ABB RobotStudio station: Abb_Robo_Challenge.rspag

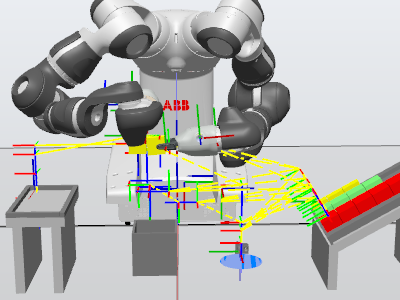
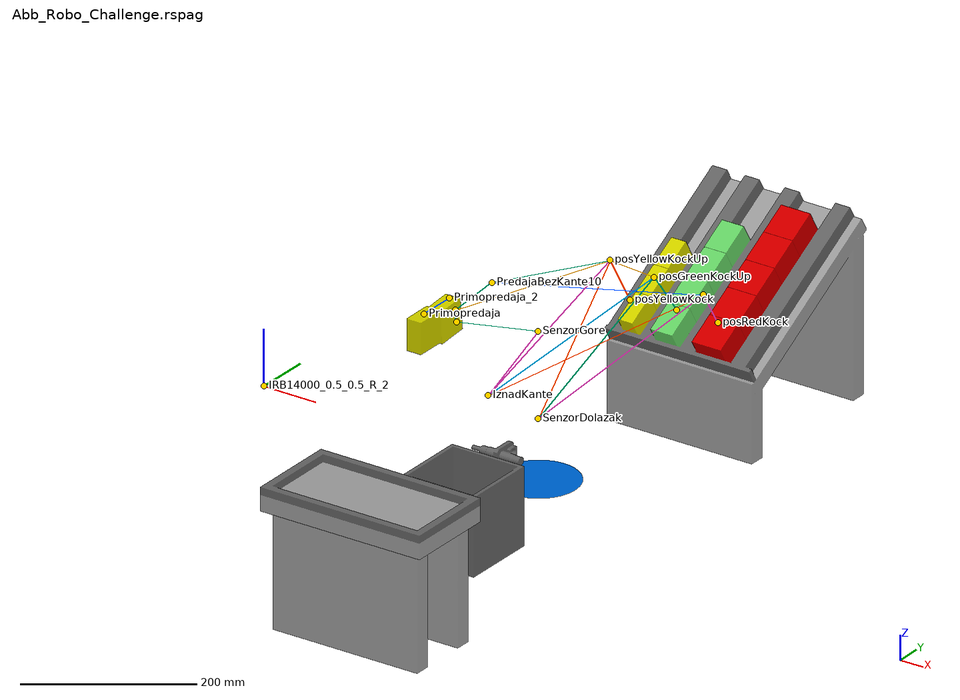
[picture v1: parts stored in the station drawn from their meshes, with robot base, taught points and paths (robot models come from the ABB library and are not in the file)]
--- station ---
Station Solution3 (saved by RobotStudio 22.3.10190.2)
Controller IRB14000, task T_ROB_L: task frame (RAPID world) sits at (0, 0, 100) mm in the station
Controller IRB14000, task T_ROB_R: task frame (RAPID world) sits at (0, 0, 100) mm in the station
Controller IRB14000
  mechanical unit ROB_R: IRB14000_0.5_0.5_R_2, 6 joints, base frame (0, 0, 0) mm
  mechanical unit ROB_R_7: IRB14000_0.5_0.5_R_2, 1 joints, base frame (0, 0, 0) mm
  mechanical unit ROB_L: IRB14000_0.5_0.5_L_2, 6 joints, base frame (0, 0, 0) mm
  mechanical unit ROB_L_7: IRB14000_0.5_0.5_L_2, 1 joints, base frame (0, 0, 0) mm
Layout (positions relative to the parent item):
  - Smart_Gripper_Servo_One_Vacuum_Fingers [mechanism, from Tools\ABB_Smart_Gripper_Servo_One_Vacuum_Fingers.rslib] at (280.99, 90.09, 293.14) mm, rotated rx 94.8 ry -1.33 rz -0.03 deg; joint values [0.0203] (rad or m)
  - Smart_Gripper_Servo_One_Vacuum_Camera_Fingers [mechanism, from Tools\ABB_Smart_Gripper_Servo_One_Vacuum_Camera_Fingers.rslib] at (319.77, -68.88, 368.32) mm, rotated rx 40.81 ry 90 rz -139.19 deg; joint values [0] (rad or m)
  - Senzor_Metala [part] at (250, 150, 15) mm, rotated rx 0 ry 0 rz 180 deg, size 65 x 32 x 27 mm
  - Mesto za testiranje [part] at (275, 150, 0) mm, size 100 x 99.5 x 0 mm
  - Rampa sa kutijama [graphiccomponentgroup]
    - Part_20 [part] at (374.5, 471.2, 184.6) mm, rotated rx 30 ry 0 rz 0 deg, size 40 x 40 x 40 mm
    - Part_1 [part] at (250, 320, 0) mm, size 200 x 20 x 100 mm
    - Part_2 [part] at (250, 520, 0) mm, size 200 x 20 x 200 mm
    - Part_3 [part], size 200 x 226.5 x 142.3 mm
    - Part_4 [part], size 200 x 14.3 x 19.8 mm
    - Part_5 [part], size 20 x 217.8 x 137.3 mm
    - Part_6 [part] at (45, 0, 0) mm, size 20 x 217.8 x 137.3 mm
    - Part_7 [part] at (100, 0, 0) mm, size 20 x 217.8 x 137.3 mm
    - Part_8 [part] at (170, 0, 0) mm, size 20 x 217.8 x 137.3 mm
    - Part_10 [part] at (292.5, 364.68, 123.1) mm, rotated rx 30 ry 0 rz 0 deg, size 20 x 40 x 40 mm
    - Part_11 [part] at (292.5, 400.18, 143.6) mm, rotated rx 30 ry 0 rz 0 deg, size 20 x 40 x 40 mm
    - Part_12 [part] at (317.5, 329.17, 102.6) mm, rotated rx 30 ry 0 rz 0 deg, size 30 x 40 x 40 mm
    - Part_13 [part] at (317.5, 364.68, 123.1) mm, rotated rx 30 ry 0 rz 0 deg, size 30 x 40 x 40 mm
    - Part_14 [part] at (317.5, 400.18, 143.6) mm, rotated rx 30 ry 0 rz 0 deg, size 30 x 40 x 40 mm
    - Part_15 [part] at (374.5, 329.17, 102.6) mm, rotated rx 30 ry 0 rz 0 deg, size 40 x 40 x 40 mm
    - Part_16 [part] at (374.5, 364.68, 123.1) mm, rotated rx 30 ry 0 rz 0 deg, size 40 x 40 x 40 mm
    - Part_17 [part] at (374.5, 400.18, 143.6) mm, rotated rx 30 ry 0 rz 0 deg, size 40 x 40 x 40 mm
    - Part_18 [part] at (317.5, 435.69, 164.1) mm, rotated rx 30 ry 0 rz 0 deg, size 30 x 40 x 40 mm
    - Part_19 [part] at (374.5, 435.69, 164.1) mm, rotated rx 30 ry 0 rz 0 deg, size 40 x 40 x 40 mm
    - Part_9 [part] at (290.75, -67.71, 300.19) mm, rotated rx -85.2 ry -1.33 rz -0.03 deg, size 20 x 40 x 40 mm
  - Paleta [graphiccomponentgroup]
    - Part_31 [part] at (450, -340, 170) mm, size 10 x 100 x 10 mm
    - Part_21 [part] at (250, -340, 0) mm, size 200 x 20 x 150 mm
    - Part_22 [part] at (250, -260, 0) mm, size 200 x 20 x 150 mm
    - Part_25 [part] at (240, -350, 170) mm, size 220 x 10 x 10 mm
    - Part_26 [part] at (240, -240, 170) mm, size 220 x 10 x 10 mm
    - Part_27 [part] at (240, -350, 150) mm, size 220 x 120 x 20 mm
    - Part_28 [part] at (240, -340, 170) mm, size 10 x 100 x 10 mm
  - Mesto za odlaganje [part], size 100 x 100 x 100 mm
  - Part_23 [part] at (292.5, 329.17, 102.6) mm, rotated rx 30 ry 0 rz 0 deg, size 20 x 40 x 40 mm
  - Pomocni_Desni [part] at (292.31, -67.5, 304.23) mm, rotated rx 180 ry 0 rz 0 deg, size 20 x 40 x 40 mm
  - IRB14000_0.5_0.5_2 [mechanism, from Robots\IRB14000_0.5_0.5__01.rslib] at (0, 0, 100) mm
  - IRB14000_0.5_0.5_R_2 [mechanism, from Robots\IRB14000_0.5_0.5__01.rslib] at (0, 0, 100) mm; joint values [1.4853, -1.6274, -1.2622, 0.7026, -0.8535, 2.2173, -1.4411] (rad or m)
  - IRB14000_0.5_0.5_L_2 [mechanism, from Robots\IRB14000_0.5_0.5__01.rslib] at (0, 0, 100) mm; joint values [-1.2905, -2.4868, 1.2641, 0.7988, -4.7194, 1.3107, 3.1478] (rad or m)
Attachment: Part_8 is attached to Part_7
Attachment: Part_7 is attached to Part_6
Attachment: Part_6 is attached to Part_5
Attachment: Part_5 is attached to Part_4
Attachment: Part_4 is attached to Part_3
Attachment: Part_3 is attached to Part_2
Attachment: Part_2 is attached to Part_1
Attachment: Part_10 is attached to Part_4
Attachment: Part_11 is attached to Part_4
Attachment: Part_12 is attached to Part_4
Attachment: Part_13 is attached to Part_4
Attachment: Part_14 is attached to Part_4
Attachment: Part_15 is attached to Part_4
Attachment: Part_16 is attached to Part_4
Attachment: Part_17 is attached to Part_4
Attachment: Part_18 is attached to Part_4
Attachment: Part_19 is attached to Part_4
Attachment: Part_20 is attached to Part_4
Attachment: Part_31 is attached to Part_28
Attachment: Part_28 is attached to Part_26
Attachment: Part_26 is attached to Part_25
Attachment: Part_25 is attached to Part_27
Attachment: Part_27 is attached to Part_22
Attachment: Part_22 is attached to Part_21
Attachment: Part_9 is attached to Smart_Gripper_Servo_One_Vacuum_Fingers / DownFinger
Attachment: Pomocni_Desni is attached to Pneumatic
Attachment: Smart_Gripper_Servo_One_Vacuum_Camera_Fingers is attached to IRB14000_0.5_0.5_R_2 / Link7
Attachment: Smart_Gripper_Servo_One_Vacuum_Fingers is attached to IRB14000_0.5_0.5_L_2 / Link7
Targets, tools, work objects and paths stored in the station and not in the controller backup, written as RAPID:
! task T_ROB_R
MODULE PROGRAM_R
  VAR syncident sync1;
  VAR syncident sync2;
  VAR syncident sync3;
ENDMODULE

! task T_ROB_L
MODULE PROGRAM_L
  VAR syncident sync1;
  VAR syncident sync2;
  VAR syncident sync3;
ENDMODULE

! task T_ROB_R
MODULE PROGRAM_R
  VAR syncident sync1;
  VAR syncident sync2;
ENDMODULE

! task T_ROB_L
MODULE PROGRAM_L
  VAR syncident sync1;
  VAR syncident sync2;
ENDMODULE


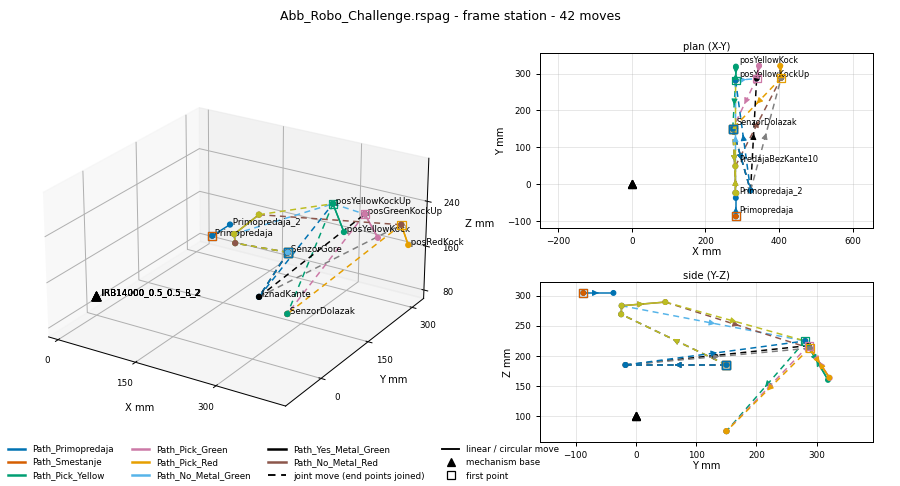
[picture p0: tool path of Abb_Robo_Challenge.rspag in frame station, 42 of 45 moves have a stored position in this frame; points joined in program order, loops and branches not executed]
--- Backups/IRB14000/RAPID/TASK1/PROGMOD/CalibData.mod ---
MODULE CalibData
    PERS tooldata Servo:=[TRUE,[[0,0,114.2],[1,0,0,0]],[0.24,[8.2,12.5,48.1],[1,0,0,0],0.00022,0.00024,0.00009]];
    PERS tooldata VaccumOne:=[TRUE,[[63.5,18.5,37.5],[0.707106781,0,0.707106781,0]],[0.24,[8.2,12.5,48.1],[1,0,0,0],0.00022,0.00024,0.00009]];
    PERS tooldata Camera:=[TRUE,[[-7.3,28.3,35.1],[0.5,-0.5,0.5,0.5]],[0.24,[8.2,12.5,48.1],[1,0,0,0],0.00022,0.00024,0.00009]];
    PERS wobjdata woKantaR:=[FALSE,TRUE,"",[[282.386,-62.26,79.768],[0.707106781,-0.707106781,0,0]],[[0,0,0],[1,0,0,0]]];
    PERS wobjdata woPreuzmi:=[FALSE,TRUE,"",[[282.386,102.74,79.768],[0.707106781,-0.707106781,0,0]],[[0,0,0],[1,0,0,0]]];
    PERS wobjdata woPaleta:=[FALSE,TRUE,"",[[250,-330.604465451,70],[1,0,0,0]],[[0,0,0],[1,0,0,0]]];
ENDMODULE

--- Backups/IRB14000/RAPID/TASK1/PROGMOD/Module1.mod ---
MODULE Module1
    PERS num br_duzina;
    PERS num br_visina;
    PERS num pomeraj;



       !  !!!!!!!!!!!!!!!!!!!!!!!!!!!!!!!!

    CONST robtarget posHome:=[[54.845252741,-184.443859011,238.96369283],[0.12531745,-0.225816146,-0.031964186,-0.965546941],[0,0,0,4],[-101.964427132,9E+09,9E+09,9E+09,9E+09,9E+09]];
    CONST robtarget posKodKante:=[[0,-100,-20],[1,0,0,0],[0,0,0,0],[-101.964427132,9E+09,9E+09,9E+09,9E+09,9E+09]];
    CONST robtarget posKodKante_3:=[[0,0,-20],[1,0,0,0],[0,0,0,0],[-101.964427132,9E+09,9E+09,9E+09,9E+09,9E+09]];
    CONST robtarget posKodKante_2:=[[0,0,0],[1,0,0,0],[0,0,0,0],[-101.964427132,9E+09,9E+09,9E+09,9E+09,9E+09]];
    CONST robtarget posTranzicija:=[[-0.118930441,-20.052950344,-210.115205223],[1,-0.000000095,-0.000000108,0.000000158],[1,-1,2,4],[-147.412404821,9E+09,9E+09,9E+09,9E+09,9E+09]];
    CONST robtarget posIznadSenzora:=[[-8.495,34.489,-98.444458216],[1,0,0,0],[1,-1,2,4],[-147.412404821,9E+09,9E+09,9E+09,9E+09,9E+09]];
    CONST robtarget posTranzicija_2:=[[-0.118939501,-5.052946544,-190.115208073],[1,-0.000000095,-0.000000108,0.000000158],[1,-1,2,4],[-147.412404821,9E+09,9E+09,9E+09,9E+09,9E+09]];

    VAR robtarget posTranzicija_3:=[[-0.118914221,-85.052946544,-170.115192873],[0.500000023,-0.500000086,0.49999982,0.500000072],[1,-1,-1,4],[-147.412404821,9E+09,9E+09,9E+09,9E+09,9E+09]];
    VAR robtarget poz_iznad_palete_2:=[[20,9.582041834,90],[0,-0.707106781,0.707106781,0],[0,0,-2,4],[-170.196454308,9E+09,9E+09,9E+09,9E+09,9E+09]];
    VAR robtarget poz_iznad_palete:=[[20.00,9.99,-12.75],[2.11141E-05,0.707095,-0.707119,-9.2686E-07],[1,0,-2,4],[-170.196,9E+09,9E+09,9E+09,9E+09,9E+09]];
    CONST robtarget Primopredaja:=[[-0.118901581,-125.052946544,-190.115185273],[0.707106714,-0.707106848,-0.000000188,0.000000035],[1,-1,-1,4],[-147.412404821,9E+09,9E+09,9E+09,9E+09,9E+09]];
    CONST robtarget Primopredaja_2:=[[-0.118912401,-125.052956019,-140.115185273],[0.707106714,-0.707106848,-0.000000188,0.000000035],[1,-1,-1,4],[-147.412404821,9E+09,9E+09,9E+09,9E+09,9E+09]];


    PROC Path_Primopredaja()

        MoveJ Primopredaja,v500,z50,VaccumOne\WObj:=woPreuzmi;
        MoveL Primopredaja_2,v50,fine,VaccumOne\WObj:=woPreuzmi;
        g_VacuumOn1;
        WaitSyncTask \InPos, sync1,task_list;


        WaitSyncTask sync2,task_list;
        WaitTime\InPos,0.1;
        WaitSyncTask sync3,task_list;

    ENDPROC
    PROC Path_Smestanje()
        poz_iznad_palete_2:=[[20+br_duzina*43,9.99+pomeraj,90+br_visina*42],[0,-0.707106781,0.707106781,0],[0,0,-2,4],[-170.196454308,9E+09,9E+09,9E+09,9E+09,9E+09]];
        !poz_iznad_palete:=[[20+br_duzina*40,10+pomeraj,45+br_visina*40],[0,-0.707106781,0.707106781,0],[1,0,-2,4],[-170.196454308,9E+09,9E+09,9E+09,9E+09,9E+09]];
        poz_iznad_palete:=[[20.00+br_duzina*43,9.99+pomeraj,-12.75+br_visina*42],[2.11141E-05,0.707095,-0.707119,-9.2686E-07],[1,0,-2,4],[-170.196,9E+09,9E+09,9E+09,9E+09,9E+09]];
        posTranzicija_3:=[[-0.118914221,-85.052946544,-170.115192873+br_visina*40],[0.500000023,-0.500000086,0.49999982,0.500000072],[1,-1,-1,4],[-147.412404821,9E+09,9E+09,9E+09,9E+09,9E+09]];


        MoveL poz_iznad_palete_2,v500,fine,VaccumOne\WObj:=woPaleta;
        MoveL poz_iznad_palete,v50,fine,VaccumOne\WObj:=woPaleta;
        WaitTime \InPos, 0.1;
        g_VacuumOff1;
        MoveL poz_iznad_palete_2,v100,fine,VaccumOne\WObj:=woPaleta;
        MoveL Primopredaja,v500,z100,VaccumOne\WObj:=woPreuzmi;
    ENDPROC
ENDMODULE

--- Backups/IRB14000/RAPID/TASK1/PROGMOD/PROGRAM_R.mod ---
MODULE PROGRAM_R

    PERS num IsMetal;
    VAR syncident sync1;
    PERS tasks task_list{2}:=[["T_ROB_L"], ["T_ROB_R"]];
    VAR syncident sync2;
    VAR syncident sync3;
    PERS bool radi;

    PROC main()
        g_Init;
        WHILE radi  DO
            Path_Primopredaja;
            IF IsMetal = 1 THEN
                g_VacuumOff1;
            ELSE
                Path_Smestanje;
            ENDIF

        ENDWHILE
    ENDPROC
ENDMODULE

--- Backups/IRB14000/RAPID/TASK2/PROGMOD/CalibData.mod ---
MODULE CalibData
    PERS tooldata Servo:=[TRUE,[[0,0,114.2],[1,0,0,0]],[0.226,[8.9,12.3,48.7],[1,0,0,0],0.00021,0.00024,0.00009]];
    PERS tooldata VaccumOne:=[TRUE,[[63.5,18.5,37.5],[0.707106781,0,0.707106781,0]],[0.226,[8.9,12.3,48.7],[1,0,0,0],0.00021,0.00024,0.00009]];
    PERS wobjdata woYellow:=[FALSE,TRUE,"",[[282.5,326.49,47.239],[0,1,0,0]],[[0,0,0],[1,0,0,0]]];
    PERS wobjdata woSenzor:=[FALSE,TRUE,"",[[250,150,-85],[0,1,0,0]],[[0,0,0],[1,0,0,0]]];
ENDMODULE

--- Backups/IRB14000/RAPID/TASK2/PROGMOD/Module1.mod ---
MODULE Module1

    PERS num IsMetal;

    CONST robtarget posHome:=[[89.387946423,156.622117957,147.913470217],[0.066010726,0.842420918,-0.111214912,0.523068661],[0,0,0,4],[101.964427132,9E+09,9E+09,9E+09,9E+09,9E+09]];
    CONST robtarget posYellowKockRanije:=[[0,18.749999999,-32.475952643],[0,0,-0.258819045,0.965925826],[-1,0,-2,4],[101.964431609,9E+09,9E+09,9E+09,9E+09,9E+09]];
    CONST robtarget posYellowKock:=[[0.02,7.64,-13.22],[0.965927,0.258817,1.54824E-05,-1.41526E-06],[-1,-2,2,4],[102.778,9E+09,9E+09,9E+09,9E+09,9E+09]];
    CONST robtarget posYellowKockPomeranje:=[[0,188.749999999,-32.475952643],[0.707106781,0,0,-0.707106781],[-1,0,-2,4],[101.964431609,9E+09,9E+09,9E+09,9E+09,9E+09]];
    CONST robtarget posYellowKockPomeranjeKodKante:=[[0,183.749999999,-32.475952643],[0,0,0.707106781,0.707106781],[-1,0,-2,4],[101.964431609,9E+09,9E+09,9E+09,9E+09,9E+09]];
    CONST robtarget posYellowKockUp:=[[-0.79,45.49,-77.87],[0.965923,0.258814,-0.00274869,-8.89019E-05],[-1,-2,2,4],[105.77,9E+09,9E+09,9E+09,9E+09,9E+09]];
    CONST robtarget SenzorDole:=[[23.88,-0.26,-60.27],[0.70711,-4.12547E-06,-1.47362E-07,0.707103],[-1,-2,3,4],[141.48,9E+09,9E+09,9E+09,9E+09,9E+09]];
    CONST robtarget SenzorDolazak:=[[23.884,-0.258,-60.279],[0.707106781,0,0,0.707106781],[-1,-2,3,4],[101.9644362,9E+09,9E+09,9E+09,9E+09,9E+09]];
    CONST robtarget posGreenKockUp:=[[56.24,39.87,-70.18],[0.964961,0.260483,0.0305117,0.00826304],[-1,-2,2,4],[102.041,9E+09,9E+09,9E+09,9E+09,9E+09]];
    CONST robtarget posGreenKock:=[[62.94,4.81,-16.31],[0.96335,0.268246,0.000869685,-0.000743491],[-1,-2,2,4],[102.163,9E+09,9E+09,9E+09,9E+09,9E+09]];
    CONST robtarget posRedKockUp:=[[123.01,38.04,-65.90],[0.965925,0.258824,1.16659E-05,7.82068E-07],[-1,-2,2,4],[101.964,9E+09,9E+09,9E+09,9E+09,9E+09]];
    CONST robtarget posRedKock:=[[120.22,5.44,-16.96],[0.962691,0.270603,-0.000479747,0.000162174],[-1,-2,2,4],[102.085,9E+09,9E+09,9E+09,9E+09,9E+09]];
    CONST robtarget SenzorTransakcije:=[[32.27,167.38,-150.279],[0.707106781,-0.707106781,0,0],[-1,-2,3,4],[101.9644362,9E+09,9E+09,9E+09,9E+09,9E+09]];
    CONST robtarget Predaja:=[[32.27,165.38,-230.279],[0.707106781,-0.707106781,0,0],[-1,-2,3,4],[101.9644362,9E+09,9E+09,9E+09,9E+09,9E+09]];
    CONST robtarget Predaja_2:=[[29.46,165.24,-255.08],[0.736071,-0.676804,0.00842612,0.00806546],[-1,-3,2,4],[105.413,9E+09,9E+09,9E+09,9E+09,9E+09]];
    CONST robtarget PredajaBezKante:=[[31.15,173.71,-268.59],[0.736045,-0.676832,0.00838831,0.00808762],[-1,-3,2,4],[105.663,9E+09,9E+09,9E+09,9E+09,9E+09]];
    CONST robtarget SenzorDolazak_2:=[[23.884,-0.258,-140.279],[0.707106781,0,0,0.707106781],[-1,-2,3,4],[101.9644362,9E+09,9E+09,9E+09,9E+09,9E+09]];
    CONST robtarget SenzorTransakcije_2:=[[32.27,167.38,-130.279],[0.707106781,-0.707106781,0,0],[-1,-2,3,4],[101.9644362,9E+09,9E+09,9E+09,9E+09,9E+09]];
    CONST robtarget IznadKante:=[[72.27,167.38,-170.279],[0.707106781,-0.707106781,0,0],[-1,-2,3,4],[101.9644362,9E+09,9E+09,9E+09,9E+09,9E+09]];
    CONST robtarget SenzorGore:=[[23.884,-0.258,-170.279],[0.707106781,0,0,0.707106781],[-1,-2,3,4],[101.9644362,9E+09,9E+09,9E+09,9E+09,9E+09]];
    CONST robtarget Predaja_12:=[[33.47,174.51,-254.40],[0.736066,-0.676809,0.00842033,0.00807085],[-1,-3,2,4],[105.403,9E+09,9E+09,9E+09,9E+09,9E+09]];
    CONST robtarget PredajaBezKante10:=[[31.05,101.22,-274.67],[0.736039,-0.676839,0.00837774,0.00808113],[-1,-3,2,4],[105.739,9E+09,9E+09,9E+09,9E+09,9E+09]];
    PROC Path_Pick_Yellow()
        g_Gripout;
        MoveJ posYellowKockUp,v500,fine,Servo\WObj:=woYellow;
        MoveL posYellowKock,v100,fine,Servo\WObj:=woYellow;
        WaitTime\InPos,0.1;
        g_Gripin;
        MoveL posYellowKockUp, v100, fine, Servo\WObj:=woYellow;
        MoveJ SenzorDolazak,v500,fine,Servo\WObj:=woSenzor;
        MoveL SenzorDole,v100,fine,Servo\WObj:=woSenzor;

        IF MetalSensor = 1 THEN
            IsMetal:=1;
        ELSE
            IsMetal := 0;
        ENDIF


        WaitTime\InPos,1;
    ENDPROC
    PROC Path_Pick_Green()
        g_Gripout;
        MoveJ posGreenKockUp,v500,fine,Servo\WObj:=woYellow;
        MoveL posGreenKock,v100,fine,Servo\WObj:=woYellow;
        WaitTime\InPos,0.1;
        g_Gripin;
        MoveL posGreenKockUp,v100,fine,Servo\WObj:=woYellow;
        MoveJ SenzorDolazak,v500,z50,Servo\WObj:=woSenzor;
        MoveL SenzorDole,v100,fine,Servo\WObj:=woSenzor;

        IF MetalSensor = 1 THEN
            IsMetal:=1;
        ELSE
            IsMetal := 0;
        ENDIF
        WaitTime\InPos,1;



    ENDPROC
    PROC Path_Pick_Red()
        g_Gripout;
        MoveJ posRedKockUp,v500,fine,Servo\WObj:=woYellow;
        MoveL posRedKock,v100,fine,Servo\WObj:=woYellow;
        WaitTime\InPos,0.1;
        g_GripIn;
        MoveL posRedKockUp,v100,fine,Servo\WObj:=woYellow;
        MoveJ SenzorDolazak,v500,fine,Servo\WObj:=woSenzor;
        MoveL SenzorDole,v100,fine,Servo\WObj:=woSenzor;

        IF MetalSensor = 1 THEN
            IsMetal:=1;
        ELSE
            IsMetal := 0;
        ENDIF



        WaitTime\InPos,1;
    ENDPROC
    PROC Path_No_Metal_Green()
        MoveJ SenzorGore,v500,z100,Servo\WObj:=woSenzor;
        MoveJ Predaja_12, v500, z100, Servo\WObj:=woSenzor;
        MoveL PredajaBezKante, v50, fine, Servo\WObj:=woSenzor;
        WaitSyncTask sync1,task_list;
        WaitSyncTask sync2,task_list;
        g_GripOut;
        WaitTime \Inpos, 0.5; !!!Jel potrebno?

        WaitSyncTask sync3,task_list;
        MoveJ posYellowKockUp,v500,fine,Servo\WObj:=woYellow;


        MoveJ posGreenKockUp,v500,fine,Servo\WObj:=woYellow;
    ENDPROC
    PROC Path_Yes_Metal_Green()
        MoveJ SenzorGore,v500,z100,Servo\WObj:=woSenzor;
        MoveJ IznadKante,v500,fine,Servo\WObj:=woSenzor;
        g_Gripout;
        WaitTime\InPos,0.2; !!Mozda previse
        MoveJ posGreenKockUp,v500,fine,Servo\WObj:=woYellow;

    ENDPROC
    PROC Path_No_Metal_Red()
        MoveJ SenzorGore,v500,z100,Servo\WObj:=woSenzor;
        MoveJ Predaja_12, v500, z100, Servo\WObj:=woSenzor;
        MoveL PredajaBezKante, v50, fine, Servo\WObj:=woSenzor;
        WaitSyncTask sync1,task_list;
        WaitSyncTask sync2,task_list;
        g_GripOut;
        WaitTime\InPos,0.5;
        MoveL PredajaBezKante10, v50, fine, Servo\WObj:=woSenzor;
        WaitSyncTask sync3,task_list;
        MoveJ posRedKockUp,v500,fine,Servo\WObj:=woYellow;
    ENDPROC
    PROC Path_Yes_Metal_Red()
        MoveJ SenzorGore,v500,z100,Servo\WObj:=woSenzor;
        MoveJ IznadKante,v500,fine,Servo\WObj:=woSenzor;
        g_Gripout;
        WaitTime\InPos,0.2;
        MoveJ posRedKockUp,v500,fine,Servo\WObj:=woYellow;
    ENDPROC
    PROC Path_No_Metal_Yellow()
        MoveJ SenzorGore,v500,z100,Servo\WObj:=woSenzor;
        MoveJ Predaja_12, v500, z100, Servo\WObj:=woSenzor;
        MoveL PredajaBezKante, v50, fine, Servo\WObj:=woSenzor;
        WaitSyncTask sync1,task_list;
        WaitSyncTask sync2,task_list;
        g_GripOut;
        WaitTime\InPos,0.5;
        MoveL PredajaBezKante10, v50, fine, Servo\WObj:=woSenzor;
        WaitSyncTask sync3,task_list;
        MoveJ posYellowKockUp,v500,fine,Servo\WObj:=woYellow;
    ENDPROC
    PROC Path_Yes_Metal_Yellow()
        MoveJ SenzorGore,v500,z100,Servo\WObj:=woSenzor;
        MoveJ IznadKante,v500,fine,Servo\WObj:=woSenzor;
        g_Gripout;
        WaitTime\InPos,0.2;
        MoveJ posYellowKockUp,v500,fine,Servo\WObj:=woYellow;
    ENDPROC


ENDMODULE

--- Backups/IRB14000/RAPID/TASK2/PROGMOD/PROGRAM_L.mod ---
MODULE PROGRAM_L

    PERS tasks task_list{2}:=[["T_ROB_L"], ["T_ROB_R"]];
    VAR syncident sync1;
    VAR syncident sync2;
    VAR syncident sync3;


    VAR num br_duzina_zute;
    VAR num br_duzina_crvene;
    VAR num br_duzina_zelene;
    VAR num br_visina_zute;
    VAR num br_visina_crvene;
    VAR num br_visina_zelene;

    PERS num br_duzina;
    PERS num br_visina;
    PERS num pomeraj;

    PERS bool radi;

    PROC main()

        VAR num zuta;
        VAR num zelena;
        VAR num crvena;
        VAR num j;
        VAR num odluka1;
        VAR num odluka2;
        VAR num odluka3;
        VAR num odluka4;
        VAR bool pp := TRUE;

        radi := TRUE;


       br_duzina_zute:=0;
       br_duzina_crvene:=0;
       br_duzina_zelene:=0;
       br_visina_zute:=0;
       br_visina_crvene:=0;
       br_visina_zelene:=0;



      WHILE pp DO
            TPReadFK odluka1, "Koliko vrsta zelite?", "1", stEmpty, "2", stEmpty, "3";

            IF odluka1 = 1 THEN
                TPReadFK odluka2, "Izaberite boju: ", "zuta", stEmpty, "zelena", stEmpty, "crvena";
                IF odluka2 = 1 THEN
                    zuta:=15;
                ELSE IF odluka2 = 3 THEN
                    zelena := 15;
                ELSE IF odluka2 = 5 THEN
                    crvena:=15;
                ENDIF
                ENDIF
                ENDIF

            ELSE IF odluka1 = 3 THEN
                TPReadFK odluka2, "Izaberite prvu boju: ", "zuta", stEmpty, "zelena", stEmpty, "crvena";
                IF odluka2 = 1 THEN
                    zuta:=15;

                    TPReadFK odluka3, "Izaberite drugu boju: ", stEmpty, stEmpty, "zelena", stEmpty, "crvena";
                    IF odluka3 = 3 THEN
                        zelena := 15;
                    ELSE IF odluka3 = 5 THEN
                        crvena:=15;
                    ENDIF
                    ENDIF
                ELSE IF odluka2 = 3 THEN
                    zelena := 15;

                    TPReadFK odluka3, "Izaberite drugu boju: ", "zuta", stEmpty, stEmpty, stEmpty, "crvena";
                    IF odluka3 = 1 THEN
                        zuta := 15;
                    ELSE IF odluka3 = 5 THEN
                        crvena:=15;
                    ENDIF
                    ENDIF
                ELSE IF odluka2 = 5 THEN
                    crvena:=15;

                    TPReadFK odluka3, "Izaberite drugu boju: ", "zuta", stEmpty, "zelena", stEmpty, stEmpty;
                    IF odluka3 = 1 THEN
                        zuta := 15;
                    ELSE IF odluka3 = 3 THEN
                        zelena:=15;
                    ENDIF
                    ENDIF
                ENDIF
                ENDIF
                ENDIF

            ELSE IF odluka1 = 5 THEN
                zuta := 15;
                zelena := 15;
                crvena := 15;
            ENDIF
            ENDIF
            ENDIF

            g_Init;
            g_GripOut;

            FOR i FROM 1 TO 3 DO
                setDO RobotActive,1;
                pomeraj := 0;
                IF zuta > 0 AND zuta<16 THEN
                    j:=0;
                    WHILE j<zuta AND  j<5 DO
                        br_duzina := br_duzina_zute;
                        br_visina := br_visina_zute;
                        Path_Pick_Yellow;
                        j := j+1;

                        IF IsMetal = 0 THEN
                            Path_No_Metal_Yellow;
                            IF br_duzina_zute = 4 THEN
                                br_duzina_zute := 0;
                                br_visina_zute := br_visina_zute + 1;
                            ELSE
                                br_duzina_zute := br_duzina_zute+1;
                            ENDIF
                        ELSE
                            Path_Yes_Metal_Yellow;
                        ENDIF

                    ENDWHILE
                    zuta:= zuta - j;
                ENDIF
                pomeraj:=pomeraj + 38;


                IF zelena>0 AND zelena<16 THEN
                   j:=0;
                    WHILE j<zelena AND  j<5 DO
                        br_duzina := br_duzina_zelene;
                        br_visina := br_visina_zelene;
                        Path_Pick_Green;
                        j := j+1;

                        IF IsMetal = 0 THEN
                            Path_No_Metal_Green;
                            IF br_duzina_zelene = 4 THEN
                                br_duzina_zelene:=0;
                                br_visina_zelene:= br_visina_zelene + 1;
                            ELSE
                                br_duzina_zelene:= br_duzina_zelene+1;
                            ENDIF
                        ELSE
                            Path_Yes_Metal_Green;
                        ENDIF

                    ENDWHILE
                    zelena:= zelena - j;
                ENDIF
                pomeraj:= pomeraj + 27;

                IF crvena>0 AND crvena<16 THEN
                    j:=0;
                    WHILE j<crvena AND  j<5 DO
                        br_duzina := br_duzina_crvene;
                        br_visina := br_visina_crvene;
                        Path_Pick_Red;
                        j := j+1;

                        IF IsMetal =0 THEN
                            Path_No_Metal_Red;
                            IF br_duzina_crvene = 4 THEN
                                br_duzina_crvene:=0;
                                br_visina_crvene:= br_visina_crvene + 1;
                            ELSE
                                br_duzina_crvene:= br_duzina_crvene+1;
                            ENDIF
                        ELSE
                            Path_Yes_Metal_Red;
                        ENDIF
                    ENDWHILE
                    crvena:= crvena - j;
                ENDIF
            ENDFOR
            radi := FALSE;
            setDO RobotActive,0;

            TPReadFK odluka4, "Da li je paleta ispraznjena?", "DA", stEmpty, stEmpty, stEmpty, "NE";
            IF odluka4 = 1 THEN
                pp := TRUE;
            ELSE
                pp := FALSE;
            ENDIF
        ENDWHILE
    ENDPROC


ENDMODULE

--- Backups/IRB14000/SYSPAR/EIO.cfg ---
EIO:CFG_1.0:6:1::
#
SYSSIG_IN:

      -Signal "Collision_Avoidance" -Action "CollAvoidance"
#
INDUSTRIAL_NETWORK:

      -Name "EtherNetIP" -Connection "Private Network" -Label "EtherNet/IP"

      -Name "DeviceNet" -Label "DeviceNet Master/Slave Network" -Address "2"
#
EIO_CROSS:

      -Name "Cross_Signal_Lamp" -Res "Signal_Lamp" -Act1 "DRV1BRAKE"
#
EIO_SIGNAL_SAFELEVEL:

      -Name "FlangePowerSafeLevel" -ActionWhenStartup "Last"

      -Name "SGcmdSafeLevel" -ActionWhenAccessible "Default"
#
ETHERNETIP_DEVICE:

      -Name "Hand_R" -StateWhenStartup "Deactivated" -VendorName "ABB"\
      -ProductName "EtherNet/IP EIP" -Label "2" -Address "192.168.125.30"\
      -VendorId 75 -ProductCode 1 -OutputAssembly 100 -InputAssembly 101\
      -InputConnectionType "POINT2POINT" -OutputSize 10 -InputSize 10\
      -O2T_RPI 10000 -T2O_RPI 10000 -ConnectionTimeoutMultiplier 2

      -Name "Hand_L" -StateWhenStartup "Deactivated" -VendorName "ABB"\
      -ProductName "EtherNet/IP EIP" -Label "1" -Address "192.168.125.40"\
      -VendorId 75 -ProductCode 1 -OutputAssembly 100 -InputAssembly 101\
      -InputConnectionType "POINT2POINT" -OutputSize 10 -InputSize 10\
      -O2T_RPI 10000 -T2O_RPI 10000 -ConnectionTimeoutMultiplier 2
#
DEVICENET_DEVICE:

      -Name "D652_10" -VendorName "ABB Robotics" -ProductName "24 VDC Unit"\
      -Address 10 -ProductCode 26 -DeviceType 7 -ConnectionType "COS"\
      -OutputSize 2 -InputSize 2
#
DEVICENET_INTERNAL_DEVICE:

      -Name "DN_Internal_Device" -VendorName "ABB Robotics"\
      -ProductName "DeviceNet Internal Slave Device"
#
ETHERNETIP_INTERNAL_DEVICE:

      -Name "EN_Internal_Device" -VendorName "ABB Robotics"\
      -ProductName "EtherNet/IP Internal Adapter Device"
#
EIO_SIGNAL:

      -Name "custom_DI_0" -SignalType "DI" -Device "D652_10" -DeviceMap "0"

      -Name "custom_DI_1" -SignalType "DI" -Device "D652_10" -DeviceMap "1"

      -Name "custom_DI_2" -SignalType "DI" -Device "D652_10" -DeviceMap "2"

      -Name "custom_DI_3" -SignalType "DI" -Device "D652_10" -DeviceMap "3"

      -Name "custom_DI_4" -SignalType "DI" -Device "D652_10" -DeviceMap "4"

      -Name "custom_DI_5" -SignalType "DI" -Device "D652_10" -DeviceMap "5"

      -Name "custom_DI_6" -SignalType "DI" -Device "D652_10" -DeviceMap "6"

      -Name "custom_DI_7" -SignalType "DI" -Device "D652_10" -DeviceMap "7"

      -Name "custom_DO_0" -SignalType "DO" -Device "D652_10" -DeviceMap "0"

      -Name "custom_DO_1" -SignalType "DO" -Device "D652_10" -DeviceMap "1"

      -Name "custom_DO_2" -SignalType "DO" -Device "D652_10" -DeviceMap "2"

      -Name "custom_DO_3" -SignalType "DO" -Device "D652_10" -DeviceMap "3"

      -Name "custom_DO_4" -SignalType "DO" -Device "D652_10" -DeviceMap "4"

      -Name "custom_DO_5" -SignalType "DO" -Device "D652_10" -DeviceMap "5"

      -Name "custom_DO_6" -SignalType "DO" -Device "D652_10" -DeviceMap "6"

      -Name "custom_DO_7" -SignalType "DO" -Device "D652_10" -DeviceMap "7"

      -Name "hall_sensor_joint_1" -SignalType "DI" -Device "D652_10"\
      -DeviceMap "8"

      -Name "hall_sensor_joint_2" -SignalType "DI" -Device "D652_10"\
      -DeviceMap "9"

      -Name "hall_sensor_joint_3" -SignalType "DI" -Device "D652_10"\
      -DeviceMap "11"

      -Name "hall_sensor_joint_4" -SignalType "DI" -Device "D652_10"\
      -DeviceMap "12"

      -Name "hall_sensor_joint_5" -SignalType "DI" -Device "D652_10"\
      -DeviceMap "13"

      -Name "hall_sensor_joint_6" -SignalType "DI" -Device "D652_10"\
      -DeviceMap "14"

      -Name "hall_sensor_joint_7" -SignalType "DI" -Device "D652_10"\
      -DeviceMap "10"

      -Name "hall_sensor_24V_ROB_R" -SignalType "DO" -Device "D652_10"\
      -DeviceMap "8"

      -Name "hall_sensor_24V_ROB_L" -SignalType "DO" -Device "D652_10"\
      -DeviceMap "9"

      -Name "flange_24V_ROB_R" -SignalType "DO" -Device "D652_10"\
      -DeviceMap "10" -SafeLevel "FlangePowerSafeLevel"

      -Name "flange_24V_ROB_L" -SignalType "DO" -Device "D652_10"\
      -DeviceMap "11" -SafeLevel "FlangePowerSafeLevel"

      -Name "Signal_Lamp" -SignalType "DO" -Device "D652_10" -DeviceMap "12"

      -Name "Collision_Avoidance" -SignalType "DO" -Access "All" -Default 1

      -Name "hand_CmdGripper_R" -SignalType "GO" -Device "Hand_R"\
      -Label "Hand Command Right" -DeviceMap "0-4" -Category "HandRight"\
      -Access "All" -SafeLevel "SGcmdSafeLevel"

      -Name "hand_CmdClearErr_R" -SignalType "DO" -Device "Hand_R"\
      -Label "Clear Error Right" -DeviceMap "7" -Category "HandRight"\
      -Access "All"

      -Name "hand_MaxPosition_R" -SignalType "GO" -Device "Hand_R"\
      -Label "Max Position Right" -DeviceMap "8-15" -Category "HandRight"\
      -Access "All" -Default 100

      -Name "hand_MinPosition_R" -SignalType "GO" -Device "Hand_R"\
      -Label "Min Position Right" -DeviceMap "16-23" -Category "HandRight"\
      -Access "All" -Default 50

      -Name "hand_MaxSpeed_R" -SignalType "GO" -Device "Hand_R"\
      -Label "Max Speed Right" -DeviceMap "24-31" -Category "HandRight"\
      -Access "All" -Default 200

      -Name "hand_HoldForce_R" -SignalType "GO" -Device "Hand_R"\
      -Label "Hold Force Right" -DeviceMap "40-47" -Category "HandRight"\
      -Access "All" -Default 120

      -Name "hand_CmdVacuum1_R" -SignalType "DO" -Device "Hand_R"\
      -Label "Vacuum 1 Right" -DeviceMap "48" -Category "HandRight"\
      -Access "All"

      -Name "hand_CmdVacuum2_R" -SignalType "DO" -Device "Hand_R"\
      -Label "Vacuum 2 Right" -DeviceMap "49" -Category "HandRight"\
      -Access "All"

      -Name "hand_CmdBlowoff1_R" -SignalType "DO" -Device "Hand_R"\
      -Label "BlowOff 1 Right" -DeviceMap "50" -Category "HandRight"\
      -Access "All"

      -Name "hand_CmdBlowoff2_R" -SignalType "DO" -Device "Hand_R"\
      -Label "BlowOff 2 Right" -DeviceMap "51" -Category "HandRight"\
      -Access "All"

      -Name "hand_SysState_R" -SignalType "GI" -Device "Hand_R"\
      -Label "Finger State Right" -DeviceMap "0-4" -Category "HandRight"\
      -Access "All"

      -Name "hand_SysError_R" -SignalType "GI" -Device "Hand_R"\
      -Label "Finger Error Right" -DeviceMap "32-39" -Category "HandRight"\
      -Access "All"

      -Name "hand_StatusCalibrated_R" -SignalType "DI" -Device "Hand_R"\
      -Label "Calibrated Right" -DeviceMap "5" -Category "HandRight"\
      -Access "All"

      -Name "hand_ActualPosition_R" -SignalType "GI" -Device "Hand_R"\
      -Label "Actual Position Right" -DeviceMap "8-15" -Category "HandRight"\
      -Access "All"

      -Name "hand_ActualSpeed_R" -SignalType "GI" -Device "Hand_R"\
      -Label "Actual Speed Right" -DeviceMap "16-23" -Category "HandRight"\
      -Access "All"

      -Name "hand_StatusCamLinked_R" -SignalType "DI" -Device "Hand_R"\
      -Label "Camera Connection Right" -DeviceMap "40" -Category "HandRight"\
      -Access "All"

      -Name "hand_SoftwareVersion_R" -SignalType "GI" -Device "Hand_R"\
      -Label "Software Version Right" -DeviceMap "41-47" -Category "HandRight"\
      -Access "All"

      -Name "hand_StatusVacuum1_R" -SignalType "DI" -Device "Hand_R"\
      -Label "Vacuum 1 Right Status" -DeviceMap "48" -Category "HandRight"\
      -Access "All"

      -Name "hand_StatusVacuum2_R" -SignalType "DI" -Device "Hand_R"\
      -Label "Vacuum 1 Right Status" -DeviceMap "49" -Category "HandRight"\
      -Access "All"

      -Name "hand_StatusBlowoff1_R" -SignalType "DI" -Device "Hand_R"\
      -Label "SuncTool 1 Right Status" -DeviceMap "50" -Category "HandRight"\
      -Access "All"

      -Name "hand_StatusBlowoff2_R" -SignalType "DI" -Device "Hand_R"\
      -Label "SuncTool 1 Right Status" -DeviceMap "51" -Category "HandRight"\
      -Access "All"

      -Name "hand_ActualPressure1_R" -SignalType "GI" -Device "Hand_R"\
      -Label "Vacuum pressure1 Right" -DeviceMap "64-71" -Category "HandRight"\
      -Access "All"

      -Name "hand_ActualPressure2_R" -SignalType "GI" -Device "Hand_R"\
      -Label "Vacuum pressure2 Right" -DeviceMap "72-79" -Category "HandRight"\
      -Access "All"

      -Name "hand_SecurityKey_R" -SignalType "GO" -Device "Hand_R"\
      -Label "Security key right" -DeviceMap "64-71" -Category "HandRight"\
      -Access "All"

      -Name "hand_TftPFtpMode_R" -SignalType "DI" -Device "Hand_R"\
      -Label "Hand firmware update mode" -DeviceMap "7" -Category "HandRight"\
      -Access "All"

      -Name "hand_CmdGripper_L" -SignalType "GO" -Device "Hand_L"\
      -Label "Hand Command Left" -DeviceMap "0-4" -Category "HandLeft"\
      -Access "All" -SafeLevel "SGcmdSafeLevel"

      -Name "hand_CmdClearErr_L" -SignalType "DO" -Device "Hand_L"\
      -Label "Clear Error Left" -DeviceMap "7" -Category "HandLeft"\
      -Access "All"

      -Name "hand_MaxPosition_L" -SignalType "GO" -Device "Hand_L"\
      -Label "Max Position Left" -DeviceMap "8-15" -Category "HandLeft"\
      -Access "All" -Default 100

      -Name "hand_MinPosition_L" -SignalType "GO" -Device "Hand_L"\
      -Label "Min Position Left" -DeviceMap "16-23" -Category "HandLeft"\
      -Access "All" -Default 50

      -Name "hand_MaxSpeed_L" -SignalType "GO" -Device "Hand_L"\
      -Label "Max Speed Left" -DeviceMap "24-31" -Category "HandLeft"\
      -Access "All" -Default 200

      -Name "hand_HoldForce_L" -SignalType "GO" -Device "Hand_L"\
      -Label "Hold Force Left" -DeviceMap "40-47" -Category "HandLeft"\
      -Access "All" -Default 120

      -Name "hand_CmdVacuum1_L" -SignalType "DO" -Device "Hand_L"\
      -Label "Vacuum 1 Left" -DeviceMap "48" -Category "HandLeft" -Access "All"

      -Name "hand_CmdVacuum2_L" -SignalType "DO" -Device "Hand_L"\
      -Label "Vacuum 2 Left" -DeviceMap "49" -Category "HandLeft" -Access "All"

      -Name "hand_CmdBlowoff1_L" -SignalType "DO" -Device "Hand_L"\
      -Label "BlowOff 1 Left" -DeviceMap "50" -Category "HandLeft" -Access "All"

      -Name "hand_CmdBlowoff2_L" -SignalType "DO" -Device "Hand_L"\
      -Label "BlowOff 2 Left" -DeviceMap "51" -Category "HandLeft" -Access "All"

      -Name "hand_SysState_L" -SignalType "GI" -Device "Hand_L"\
      -Label "Finger State Left" -DeviceMap "0-4" -Category "HandLeft"\
      -Access "All"

      -Name "hand_SysError_L" -SignalType "GI" -Device "Hand_L"\
      -Label "Finger Error Left" -DeviceMap "32-39" -Category "HandLeft"\
      -Access "All"

      -Name "hand_StatusCalibrated_L" -SignalType "DI" -Device "Hand_L"\
      -Label "Calibrated Left" -DeviceMap "5" -Category "HandLeft" -Access "All"

      -Name "hand_ActualPosition_L" -SignalType "GI" -Device "Hand_L"\
      -Label "Actual Position Left" -DeviceMap "8-15" -Category "HandLeft"\
      -Access "All"

      -Name "hand_ActualSpeed_L" -SignalType "GI" -Device "Hand_L"\
      -Label "Actual Speed Left" -DeviceMap "16-23" -Category "HandLeft"\
      -Access "All"

      -Name "hand_StatusCamLinked_L" -SignalType "DI" -Device "Hand_L"\
      -Label "Camera Connection Left" -DeviceMap "40" -Category "HandLeft"\
      -Access "All"

      -Name "hand_SoftwareVersion_L" -SignalType "GI" -Device "Hand_L"\
      -Label "Software Version Left" -DeviceMap "41-47" -Category "HandLeft"\
      -Access "All"

      -Name "hand_StatusVacuum1_L" -SignalType "DI" -Device "Hand_L"\
      -Label "Vacuum 1 Left Status" -DeviceMap "48" -Category "HandLeft"\
      -Access "All"

      -Name "hand_StatusVacuum2_L" -SignalType "DI" -Device "Hand_L"\
      -Label "Vacuum 1 Left Status" -DeviceMap "49" -Category "HandLeft"\
      -Access "All"

      -Name "hand_StatusBlowoff1_L" -SignalType "DI" -Device "Hand_L"\
      -Label "SuncTool 1 Left Status" -DeviceMap "50" -Category "HandLeft"\
      -Access "All"

      -Name "hand_StatusBlowoff2_L" -SignalType "DI" -Device "Hand_L"\
      -Label "SuncTool 1 Left Status" -DeviceMap "51" -Category "HandLeft"\
      -Access "All"

      -Name "hand_ActualPressure1_L" -SignalType "GI" -Device "Hand_L"\
      -Label "Vacuum pressure1 Left" -DeviceMap "64-71" -Category "HandLeft"\
      -Access "All"

      -Name "hand_ActualPressure2_L" -SignalType "GI" -Device "Hand_L"\
      -Label "Vacuum pressure2 Left" -DeviceMap "72-79" -Category "HandLeft"\
      -Access "All"

      -Name "hand_SecurityKey_L" -SignalType "GO" -Device "Hand_L"\
      -Label "Security key Left" -DeviceMap "64-71" -Category "HandLeft"\
      -Access "All"

      -Name "hand_TftPFtpMode_L" -SignalType "DI" -Device "Hand_L"\
      -Label "Hand firmware update mode" -DeviceMap "7" -Category "HandLeft"\
      -Access "All"

      -Name "MetalSensor" -SignalType "DI" -Access "All"

      -Name "RobotActive" -SignalType "DO" -Access "All"
